{attribute addProperty BoxType "EL6201-0000-0017"}
{attribute addProperty Id "Slave_19A_DI0BIT10.125145Slave_19A_DI1BIT10.125146Slave_19A_DI2BIT10.125147Slave_19A_DI3BIT10.125148Slave_19B_DI0BIT10.125149Slave_19B_DI1BIT10.125150Slave_19B_DI2BIT10.125151Slave_19B_DI3BIT10.125152"}
{attribute addProperty CRC "3079461961"}
{attribute addProperty SizeInBites "8"}
{attribute addProperty SizeInBytes "1"}
TYPE Slave_19_Inputs_B78CDC49 :
STRUCT
	{attribute addProperty Name "Slave_19A_DI0"}
	Slave_19A_DI0 : BIT;
	{attribute addProperty Name "Slave_19A_DI1"}
	Slave_19A_DI1 : BIT;
	{attribute addProperty Name "Slave_19A_DI2"}
	Slave_19A_DI2 : BIT;
	{attribute addProperty Name "Slave_19A_DI3"}
	Slave_19A_DI3 : BIT;
	{attribute addProperty Name "Slave_19B_DI0"}
	Slave_19B_DI0 : BIT;
	{attribute addProperty Name "Slave_19B_DI1"}
	Slave_19B_DI1 : BIT;
	{attribute addProperty Name "Slave_19B_DI2"}
	Slave_19B_DI2 : BIT;
	{attribute addProperty Name "Slave_19B_DI3"}
	Slave_19B_DI3 : BIT;
END_STRUCT
END_TYPE

(* stored: Version 1.2.0.0, ProductVersion 3.1.4024.9
   DUT Slave_19_Inputs_B78CDC49: Id {83588625-a5a5-4146-87be-dd2dc945516c} *)
